SYSTEM System (* System Configuration *)
  (* Version 0.0, 7/6/2026, Schneider Electric *)
  APPLICATION Hidryco_Application
    (* CLP SUBSTACAO *)
    (* CLP NEREDA *)
    (* NEREDA REACTORS *)
    (* NEREDA PROCESS - HIDRYCO *)
    (* EMERGENCY RECIPIE *)
    (* NEREDA EQUIPMENT *)
    (* NEREDA AERATION *)
    (* INFLUENT FEED *)
    (* EFFLUENT *)
    (* SLUDGE BUFFER *)
    (* METAL SALT DOSING *)
    (* SLUDGE HOLDING TANK *)
    FBS
      A3_DI32K0 : IO_DI32(pin_46CCA44197086456 := '$${PATH}A3_DI32K_WORD0', pin_0CD1E891B208CBDA := '$${PATH}A3_DI32K_WORD1', pin_36419F0327C5E289 := 'RES0.InfluentFeed.Actuators.FeedReactorPump01.LocalPanel.SafetySwitchOff', pin_EB713021CCA66C0B := 'RES0.InfluentFeed.Actuators.FeedReactorPump02.LocalPanel.SafetySwitchOff', pin_2B28AC3EFC010509 := 'RES0.InfluentFeed.Actuators.FeedReactorPump03.LocalPanel.SafetySwitchOff', pin_ECB70C50847C6B8C := 'RES0.InfluentFeed.Actuators.FeedReactorPump01.LocalPanel.RemoteSelect', pin_07613AEA5B5EA3D4 := 'RES0.InfluentFeed.Actuators.FeedReactorPump01.fbFwd.DIn', pin_255156C9E2C187C7 := 'RES0.InfluentFeed.Actuators.FeedReactorPump01.LocalPanel.ElectricCircuitFail', pin_A4FEA1DCF2974931 := 'RES0.InfluentFeed.Actuators.FeedReactorPump01.LocalPanel.MoistureDetectionPumpMS', pin_330A6B5BAE9F40D2 := 'RES0.InfluentFeed.Actuators.FeedReactorPump02.LocalPanel.RemoteSelect', pin_15A3E3BB9AE8E740 := 'RES0.InfluentFeed.Actuators.FeedReactorPump02.fbFwd.DIn', pin_6F381A44E74CF961 := 'RES0.InfluentFeed.Actuators.FeedReactorPump02.LocalPanel.ElectricCircuitFail', pin_28174C1DE6948A82 := 'RES0.InfluentFeed.Actuators.FeedReactorPump02.LocalPanel.MoistureDetectionPumpMS', pin_1BA632E0922A0983 := 'RES0.InfluentFeed.Actuators.FeedReactorPump03.LocalPanel.RemoteSelect', pin_3F9A9A7D3F756840 := 'RES0.InfluentFeed.Actuators.FeedReactorPump03.fbFwd.DIn', pin_7C7DB6F90D480DE8 := 'RES0.InfluentFeed.Actuators.FeedReactorPump03.LocalPanel.ElectricCircuitFail', pin_E8D93A7BE9BA26AB := 'RES0.InfluentFeed.Actuators.FeedReactorPump03.LocalPanel.MoistureDetectionPumpMS', pin_2C3BA8CD03BB1AD1 := 'RES0.InfluentFeed.Actuators.Mixer01.LocalPanel.PowerFb', pin_BD4DD77DC1DECA3F := 'RES0.InfluentFeed.Actuators.Mixer02.LocalPanel.PowerFb', pin_BA2C5E15436FD50A := 'RES0.InfluentFeed.Actuators.Mixer01.LocalPanel.RemoteSelect', pin_58F1D1C70BD05BBB := 'RES0.InfluentFeed.Actuators.Mixer01.fbFwd.DIn', pin_202E08C1E95489B4 := 'RES0.InfluentFeed.Actuators.Mixer01.LocalPanel.ElectricCircuitFail', pin_4D7EBC78C81E0547 := 'RES0.InfluentFeed.Actuators.Mixer01.LocalPanel.MoistureDetectionPumpMS', pin_705DA0BDD5247341 := 'RES0.InfluentFeed.Actuators.Mixer02.LocalPanel.RemoteSelect', pin_C8A2275FCD06007F := 'RES0.InfluentFeed.Actuators.Mixer02.fbFwd.DIn', pin_029A065AE8EEF4A5 := '$${PATH}A3_DI32K0_CONN');
      A4_DI32K0 : IO_DI32(pin_46CCA44197086456 := '$${PATH}A4_DI32K_WORD0', pin_0CD1E891B208CBDA := '$${PATH}A4_DI32K_WORD1', pin_21F6274CBA1014D4 := 'RES0.InfluentFeed.Actuators.Mixer02.LocalPanel.ElectricCircuitFail', pin_828C0F18BDE4203E := 'RES0.InfluentFeed.Actuators.Mixer02.LocalPanel.MoistureDetectionPumpMS', pin_9E5CF06E07A0EB03 := 'RES0.SludgeBuffer.Actuators.Pump1.LocalPanel.PowerFb', pin_36419F0327C5E289 := 'RES0.SludgeBuffer.Actuators.Pump2.LocalPanel.PowerFb', pin_EB713021CCA66C0B := 'RES0.SludgeBuffer.Actuators.Pump3.LocalPanel.PowerFb', pin_2B28AC3EFC010509 := 'RES0.SludgeBuffer.Actuators.Pump1.LocalPanel.RemoteSelect', pin_ECB70C50847C6B8C := 'RES0.SludgeBuffer.Actuators.Pump1.fbFwd.DIn', pin_4067F611C03C22ED := 'RES0.SludgeBuffer.Actuators.Pump1.LocalPanel.ElectricCircuitFail', pin_07613AEA5B5EA3D4 := 'RES0.SludgeBuffer.Actuators.Pump2.LocalPanel.RemoteSelect', pin_A4FEA1DCF2974931 := 'RES0.SludgeBuffer.Actuators.Pump2.fbFwd.DIn', pin_330A6B5BAE9F40D2 := 'RES0.SludgeBuffer.Actuators.Pump2.LocalPanel.ElectricCircuitFail', pin_341ABC323332EA3F := 'RES0.SludgeBuffer.Actuators.Pump3.LocalPanel.RemoteSelect', pin_6F381A44E74CF961 := 'RES0.SludgeBuffer.Actuators.Pump3.fbFwd.DIn', pin_28174C1DE6948A82 := 'RES0.SludgeBuffer.Actuators.Pump3.LocalPanel.ElectricCircuitFail', pin_7C7DB6F90D480DE8 := 'RES0.Reactor1.Actuators.VentAerationGridValve_AV4x107.fbOpen.DIn', pin_E8D93A7BE9BA26AB := 'RES0.Reactor1.Actuators.VentAerationGridValve_AV4x107.fbClose.DIn', pin_2C3BA8CD03BB1AD1 := 'RES0.Reactor1.Actuators.AirFillValveSludgeDischarge_AV4x171.fbOpen.DIn', pin_BD4DD77DC1DECA3F := 'RES0.Reactor1.Actuators.AirFillValveSludgeDischarge_AV4x171.fbClose.DIn', pin_BA2C5E15436FD50A := 'RES0.Reactor1.Actuators.VentSludgeGridValve_AV4x172.fbOpen.DIn', pin_2DD13C1C321F4353 := 'RES0.Reactor1.Actuators.VentSludgeGridValve_AV4x172.fbClose.DIn', pin_58F1D1C70BD05BBB := 'RES0.Reactor1.Actuators.FeedValve_AV4x101.fbOpen.DIn', pin_202E08C1E95489B4 := 'RES0.Reactor1.Actuators.FeedValve_AV4x101.fbClose.DIn', pin_4D7EBC78C81E0547 := 'RES0.Reactor1.Actuators.LowerLevelValve_AV4x102.fbOpen.DIn', pin_705DA0BDD5247341 := 'RES0.Reactor1.Actuators.LowerLevelValve_AV4x102.fbClose.DIn', pin_3B4E2202D2B578AA := 'RES0.Reactor1.Actuators.DischargeValve_AV4x103.fbOpen.DIn', pin_C8A2275FCD06007F := 'RES0.Reactor1.Actuators.DischargeValve_AV4x103.fbClose.DIn', pin_029A065AE8EEF4A5 := 'RES0.A3_DI32K0.A3_DI32K0_CONN');
      A5_DI32K0 : IO_DI32(pin_46CCA44197086456 := '$${PATH}A5_DI32K_WORD0', pin_0CD1E891B208CBDA := '$${PATH}A5_DI32K_WORD1', pin_21F6274CBA1014D4 := 'RES0.Reactor2.Actuators.VentAerationGridValve_AV4x107.fbOpen.DIn', pin_828C0F18BDE4203E := 'RES0.Reactor2.Actuators.VentAerationGridValve_AV4x107.fbClose.DIn', pin_9E5CF06E07A0EB03 := 'RES0.Reactor2.Actuators.AirFillValveSludgeDischarge_AV4x171.fbOpen.DIn', pin_36419F0327C5E289 := 'RES0.Reactor2.Actuators.AirFillValveSludgeDischarge_AV4x171.fbClose.DIn', pin_EB713021CCA66C0B := 'RES0.Reactor2.Actuators.VentSludgeGridValve_AV4x172.fbOpen.DIn', pin_2B28AC3EFC010509 := 'RES0.Reactor2.Actuators.VentSludgeGridValve_AV4x172.fbClose.DIn', pin_772061FB1EC77CFC := 'RES0.Reactor2.Actuators.FeedValve_AV4x101.fbOpen.DIn', pin_ECB70C50847C6B8C := 'RES0.Reactor2.Actuators.FeedValve_AV4x101.fbClose.DIn', pin_4067F611C03C22ED := 'RES0.Reactor2.Actuators.LowerLevelValve_AV4x102.fbOpen.DIn', pin_07613AEA5B5EA3D4 := 'RES0.Reactor2.Actuators.LowerLevelValve_AV4x102.fbClose.DIn', pin_255156C9E2C187C7 := 'RES0.Reactor2.Actuators.DischargeValve_AV4x103.fbOpen.DIn', pin_A4FEA1DCF2974931 := 'RES0.Reactor2.Actuators.DischargeValve_AV4x103.fbClose.DIn', pin_15A3E3BB9AE8E740 := 'RES0.SludgeBuffer.Actuators.ValveBuffer.fbOpen.DIn', pin_6F381A44E74CF961 := 'RES0.SludgeBuffer.Actuators.ValveBuffer.fbClose.DIn', pin_28174C1DE6948A82 := 'RES0.SludgeBuffer.Actuators.ValveInfeed.fbOpen.DIn', pin_1BA632E0922A0983 := 'RES0.SludgeBuffer.Actuators.ValveInfeed.fbClose.DIn', pin_2C3BA8CD03BB1AD1 := 'RES0.InfluentFeed.Sensors.LevelSwitchInfluentBuffer.pv.DIn', pin_BD4DD77DC1DECA3F := 'RES0.Reactor1.Actuators.AerationBlockValve_AV4x170.fbOpen.DIn', pin_BA2C5E15436FD50A := 'RES0.Reactor1.Actuators.AerationBlockValve_AV4x170.fbClose.DIn', pin_2DD13C1C321F4353 := 'RES0.Reactor2.Actuators.AerationBlockValve_AV4x170.fbOpen.DIn', pin_58F1D1C70BD05BBB := 'RES0.Reactor2.Actuators.AerationBlockValve_AV4x170.fbClose.DIn', pin_029A065AE8EEF4A5 := 'RES0.A3_DI32K0.A3_DI32K0_CONN', pin_330A6B5BAE9F40D2 := 'RES0.SludgeBuffer.Actuators.ValveSupernatantReturn.fbOpen.DIn', pin_341ABC323332EA3F := 'RES0.SludgeBuffer.Actuators.ValveSupernatantReturn.fbClose.DIn', pin_23FCAB00EAAA7E55 := 'RES0.SludgeBuffer.Actuators.ValveTank2.fbOpen.DIn', pin_3F9A9A7D3F756840 := 'RES0.SludgeBuffer.Actuators.ValveTank2.fbClose.DIn', pin_7C7DB6F90D480DE8 := 'RES0.SludgeBuffer.Actuators.ValveTank1.fbOpen.DIn', pin_E8D93A7BE9BA26AB := 'RES0.SludgeBuffer.Actuators.ValveTank1.fbClose.DIn');
      A6_DI32K0 : IO_DI32(pin_46CCA44197086456 := '$${PATH}A6_DI32K_WORD0', pin_0CD1E891B208CBDA := '$${PATH}A6_DI32K_WORD1', pin_029A065AE8EEF4A5 := 'RES0.A3_DI32K0.A3_DI32K0_CONN');
      A7_DQ32TK0 : IO_DQ32(pin_302C3F69182ABC91 := '$${PATH}A7_DQ32TK_WORD0', pin_449EC30B868089F7 := '$${PATH}A7_DQ32TK_WORD1', pin_9A3A1A81B7B6D445 := 'RES0.InfluentFeed.Actuators.FeedReactorPump01.cmdFwd.DOut', pin_574F19B312039273 := 'RES0.InfluentFeed.Actuators.FeedReactorPump01.LocalPanel.ResetError_ATV', pin_289462D1695B79B9 := 'RES0.InfluentFeed.Actuators.FeedReactorPump02.cmdFwd.DOut', pin_312C400F6E937723 := 'RES0.InfluentFeed.Actuators.FeedReactorPump02.LocalPanel.ResetError_ATV', pin_3BE637AB2D7945FF := 'RES0.InfluentFeed.Actuators.FeedReactorPump03.cmdFwd.DOut', pin_22A55DF5D197312F := 'RES0.InfluentFeed.Actuators.FeedReactorPump03.LocalPanel.ResetError_ATV', pin_8561E9473423D106 := 'RES0.InfluentFeed.Actuators.Mixer01.cmdFwd.DOut', pin_22A9D026EB73BE1F := 'RES0.InfluentFeed.Actuators.Mixer01.LocalPanel.ResetError_ATV', pin_FA96DB2F4BA1237E := 'RES0.InfluentFeed.Actuators.Mixer02.cmdFwd.DOut', pin_29C78CF381382FF2 := 'RES0.InfluentFeed.Actuators.Mixer02.LocalPanel.ResetError_ATV', pin_29CEA3759F3752DE := 'RES0.SludgeBuffer.Actuators.Pump1.cmdFwd.DOut', pin_886E7CBF7859CEF7 := 'RES0.SludgeBuffer.Actuators.Pump1.LocalPanel.ResetError_ATV', pin_FD4664BC008BF5D6 := 'RES0.SludgeBuffer.Actuators.Pump2.cmdFwd.DOut', pin_33252EF2B10EEA13 := 'RES0.SludgeBuffer.Actuators.Pump2.LocalPanel.ResetError_ATV', pin_0AA04E78B7312E60 := 'RES0.SludgeBuffer.Actuators.Pump3.cmdFwd.DOut', pin_753BEBC4FB000D5B := 'RES0.SludgeBuffer.Actuators.Pump3.LocalPanel.ResetError_ATV', pin_9E16F3DA85027DF7 := 'RES0.Reactor1.Actuators.VentAerationGridValve_AV4x107.cmdOpen.DOut', pin_3452F813357567DB := 'RES0.Reactor1.Actuators.VentAerationGridValve_AV4x107.cmdClose.DOut', pin_19CF596687475EFF := 'RES0.Reactor1.Actuators.AirFillValveSludgeDischarge_AV4x171.cmdOpen.DOut', pin_894AD674E7043530 := 'RES0.Reactor1.Actuators.AirFillValveSludgeDischarge_AV4x171.cmdClose.DOut', pin_4C1794B9AC53DE50 := 'RES0.Reactor1.Actuators.VentSludgeGridValve_AV4x172.cmdOpen.DOut', pin_B27C16F31DA61BFA := 'RES0.Reactor1.Actuators.VentSludgeGridValve_AV4x172.cmdClose.DOut', pin_6AEF80E82895335D := 'RES0.Reactor1.Actuators.FeedValve_AV4x101.cmdOpen.DOut', pin_4CE944D399950301 := 'RES0.Reactor1.Actuators.FeedValve_AV4x101.cmdClose.DOut', pin_4A5E1556A870DE8E := 'RES0.Reactor1.Actuators.LowerLevelValve_AV4x102.cmdOpen.DOut', pin_BB019F781B1BA10A := 'RES0.Reactor1.Actuators.LowerLevelValve_AV4x102.cmdClose.DOut', pin_86F66632C3A9C16C := 'RES0.Reactor1.Actuators.DischargeValve_AV4x103.cmdOpen.DOut', pin_B6D2486BB09D13CD := 'RES0.Reactor1.Actuators.DischargeValve_AV4x103.cmdClose.DOut', pin_51993B782C6727EF := 'RES0.Reactor2.Actuators.VentAerationGridValve_AV4x107.cmdOpen.DOut', pin_C59E5F7297A9D375 := 'RES0.Reactor2.Actuators.VentAerationGridValve_AV4x107.cmdClose.DOut', pin_713D841585687888 := 'RES0.Reactor2.Actuators.AirFillValveSludgeDischarge_AV4x171.cmdOpen.DOut', pin_F178B2FCFCB541E9 := 'RES0.Reactor2.Actuators.AirFillValveSludgeDischarge_AV4x171.cmdClose.DOut', pin_4CB528AC475AE599 := 'RES0.A3_DI32K0.A3_DI32K0_CONN');
      A8_DQ32TK0 : IO_DQ32(pin_302C3F69182ABC91 := '$${PATH}A8_DQ32TK_WORD0', pin_449EC30B868089F7 := '$${PATH}A8_DQ32TK_WORD1', pin_9A3A1A81B7B6D445 := 'RES0.Reactor2.Actuators.VentSludgeGridValve_AV4x172.cmdOpen.DOut', pin_574F19B312039273 := 'RES0.Reactor2.Actuators.VentSludgeGridValve_AV4x172.cmdClose.DOut', pin_289462D1695B79B9 := 'RES0.Reactor2.Actuators.FeedValve_AV4x101.cmdOpen.DOut', pin_312C400F6E937723 := 'RES0.Reactor2.Actuators.FeedValve_AV4x101.cmdClose.DOut', pin_3BE637AB2D7945FF := 'RES0.Reactor2.Actuators.LowerLevelValve_AV4x102.cmdOpen.DOut', pin_22A55DF5D197312F := 'RES0.Reactor2.Actuators.LowerLevelValve_AV4x102.cmdClose.DOut', pin_8561E9473423D106 := 'RES0.Reactor2.Actuators.DischargeValve_AV4x103.cmdOpen.DOut', pin_22A9D026EB73BE1F := 'RES0.Reactor2.Actuators.DischargeValve_AV4x103.cmdClose.DOut', pin_29CEA3759F3752DE := 'RES0.SludgeBuffer.Actuators.ValveBuffer.cmdOpen.DOut', pin_886E7CBF7859CEF7 := 'RES0.SludgeBuffer.Actuators.ValveBuffer.cmdClose.DOut', pin_FD4664BC008BF5D6 := 'RES0.SludgeBuffer.Actuators.ValveInfeed.cmdOpen.DOut', pin_33252EF2B10EEA13 := 'RES0.SludgeBuffer.Actuators.ValveInfeed.cmdClose.DOut', pin_19CF596687475EFF := 'RES0.Reactor1.Actuators.AerationBlockValve_AV4x170.cmdOpen.DOut', pin_894AD674E7043530 := 'RES0.Reactor1.Actuators.AerationBlockValve_AV4x170.cmdClose.DOut', pin_4C1794B9AC53DE50 := 'RES0.Reactor2.Actuators.AerationBlockValve_AV4x170.cmdOpen.DOut', pin_B27C16F31DA61BFA := 'RES0.Reactor2.Actuators.AerationBlockValve_AV4x170.cmdClose.DOut', pin_4CB528AC475AE599 := 'RES0.A3_DI32K0.A3_DI32K0_CONN', pin_FA96DB2F4BA1237E := 'RES0.SludgeBuffer.Actuators.ValveSupernatantReturn.cmdOpen.DOut', pin_29C78CF381382FF2 := 'RES0.SludgeBuffer.Actuators.ValveSupernatantReturn.cmdClose.DOut', pin_3452F813357567DB := 'RES0.SludgeBuffer.Actuators.ValveTank1.cmdClose.DOut', pin_9E16F3DA85027DF7 := 'RES0.SludgeBuffer.Actuators.ValveTank1.cmdOpen.DOut', pin_0AA04E78B7312E60 := 'RES0.SludgeBuffer.Actuators.ValveTank2.cmdOpen.DOut', pin_753BEBC4FB000D5B := 'RES0.SludgeBuffer.Actuators.ValveTank2.cmdClose.DOut');
      SUB_A3_DI32K0 : IO_DI32(pin_46CCA44197086456 := '$${PATH}SUB_A3_DI32K_WORD0', pin_0CD1E891B208CBDA := '$${PATH}SUB_A3_DI32K_WORD1', pin_23FCAB00EAAA7E55 := 'RES0.Aerator.Actuators.V4603.LocalPanel.PowerFb', pin_3F9A9A7D3F756840 := 'RES0.Aerator.Actuators.V4604.LocalPanel.PowerFb', pin_029A065AE8EEF4A5 := '$${PATH}SUB_A3_DI32K0_CONN');
      SUB_A4_DI32K0 : IO_DI32(pin_46CCA44197086456 := '$${PATH}SUB_A4_DI32K_WORD0', pin_0CD1E891B208CBDA := '$${PATH}SUB_A4_DI32K_WORD1', pin_3B4E2202D2B578AA := 'RES0.Aerator.Actuators.V4601.LocalPanel.PowerFb', pin_C8A2275FCD06007F := 'RES0.Aerator.Actuators.V4602.LocalPanel.PowerFb', pin_029A065AE8EEF4A5 := 'RES0.SUB_A3_DI32K0.SUB_A3_DI32K0_CONN');
      SUB_A6_DI32K0 : IO_DI32(pin_46CCA44197086456 := '$${PATH}SUB_A6_DI32K_WORD0', pin_0CD1E891B208CBDA := '$${PATH}SUB_A6_DI32K_WORD1', pin_255156C9E2C187C7 := 'RES0.Aerator.Actuators.AV46_001.fbOpen.DIn', pin_A4FEA1DCF2974931 := 'RES0.Aerator.Actuators.AV46_001.fbClose.DIn', pin_330A6B5BAE9F40D2 := 'RES0.Aerator.Actuators.AV46_002.fbOpen.DIn', pin_341ABC323332EA3F := 'RES0.Aerator.Actuators.AV46_002.fbClose.DIn', pin_15A3E3BB9AE8E740 := 'RES0.Aerator.Actuators.AV46_003.fbOpen.DIn', pin_6F381A44E74CF961 := 'RES0.Aerator.Actuators.AV46_003.fbClose.DIn', pin_28174C1DE6948A82 := 'RES0.Aerator.Actuators.AV46_012.fbOpen.DIn', pin_1BA632E0922A0983 := 'RES0.Aerator.Actuators.AV46_012.fbClose.DIn', pin_23FCAB00EAAA7E55 := 'RES0.Aerator.Actuators.AV46_022.fbOpen.DIn', pin_3F9A9A7D3F756840 := 'RES0.Aerator.Actuators.AV46_022.fbClose.DIn', pin_7C7DB6F90D480DE8 := 'RES0.Aerator.Actuators.AV46_032.fbOpen.DIn', pin_E8D93A7BE9BA26AB := 'RES0.Aerator.Actuators.AV46_032.fbClose.DIn', pin_2C3BA8CD03BB1AD1 := 'RES0.Aerator.Actuators.AV46_042.fbOpen.DIn', pin_BD4DD77DC1DECA3F := 'RES0.Aerator.Actuators.AV46_042.fbClose.DIn', pin_029A065AE8EEF4A5 := 'RES0.SUB_A3_DI32K0.SUB_A3_DI32K0_CONN');
      SUB_A8_DQ32TK0 : IO_DQ32(pin_302C3F69182ABC91 := '$${PATH}SUB_A8_DQ32TK_WORD0', pin_449EC30B868089F7 := '$${PATH}SUB_A8_DQ32TK_WORD1', pin_19CF596687475EFF := 'RES0.Aerator.Actuators.AV46_001.cmdOpen.DOut', pin_894AD674E7043530 := 'RES0.Aerator.Actuators.AV46_001.cmdClose.DOut', pin_4C1794B9AC53DE50 := 'RES0.Aerator.Actuators.AV46_002.cmdOpen.DOut', pin_B27C16F31DA61BFA := 'RES0.Aerator.Actuators.AV46_002.cmdClose.DOut', pin_6AEF80E82895335D := 'RES0.Aerator.Actuators.AV46_003.cmdOpen.DOut', pin_4CE944D399950301 := 'RES0.Aerator.Actuators.AV46_003.cmdClose.DOut', pin_4A5E1556A870DE8E := 'RES0.Aerator.Actuators.AV46_012.cmdOpen.DOut', pin_BB019F781B1BA10A := 'RES0.Aerator.Actuators.AV46_012.cmdClose.DOut', pin_86F66632C3A9C16C := 'RES0.Aerator.Actuators.AV46_022.cmdOpen.DOut', pin_B6D2486BB09D13CD := 'RES0.Aerator.Actuators.AV46_022.cmdClose.DOut', pin_51993B782C6727EF := 'RES0.Aerator.Actuators.AV46_032.cmdOpen.DOut', pin_C59E5F7297A9D375 := 'RES0.Aerator.Actuators.AV46_032.cmdClose.DOut', pin_713D841585687888 := 'RES0.Aerator.Actuators.AV46_042.cmdOpen.DOut', pin_F178B2FCFCB541E9 := 'RES0.Aerator.Actuators.AV46_042.cmdClose.DOut', pin_4CB528AC475AE599 := 'RES0.SUB_A3_DI32K0.SUB_A3_DI32K0_CONN');
      V4601_STS0 : IO_DI32(pin_46CCA44197086456 := '$${PATH}V4601_STATUS', pin_0CD1E891B208CBDA := '$${PATH}V4601_FAULT', pin_029A065AE8EEF4A5 := '$${PATH}V4601_CONN', pin_21F6274CBA1014D4 := 'RES0.Aerator.Actuators.V4601.LocalPanel.RemoteSelect', pin_828C0F18BDE4203E := 'RES0.Aerator.Actuators.V4601.fbFwd.DIn', pin_36419F0327C5E289 := 'RES0.Aerator.Actuators.V4601.LocalPanel.FrequencyInverterFail', pin_4067F611C03C22ED := 'RES0.Aerator.Actuators.V4601.LocalPanel.AtvReady');
      V4601_CMD0 : IO_DQ32(pin_302C3F69182ABC91 := '$${PATH}V4601_CMD_WORD', pin_449EC30B868089F7 := '$${PATH}V4601_WORD1_NAO_USADA', pin_9A3A1A81B7B6D445 := 'RES0.Aerator.Actuators.V4601.cmdFwd.DOut', pin_289462D1695B79B9 := 'RES0.Aerator.Actuators.V4601.LocalPanel.ResetError_ATV');
      V4602_STS0 : IO_DI32(pin_46CCA44197086456 := '$${PATH}V4602_STATUS', pin_0CD1E891B208CBDA := '$${PATH}V4602_FAULT', pin_029A065AE8EEF4A5 := '$${PATH}V4602_CONN', pin_21F6274CBA1014D4 := 'RES0.Aerator.Actuators.V4602.LocalPanel.RemoteSelect', pin_828C0F18BDE4203E := 'RES0.Aerator.Actuators.V4602.fbFwd.DIn', pin_36419F0327C5E289 := 'RES0.Aerator.Actuators.V4602.LocalPanel.FrequencyInverterFail', pin_4067F611C03C22ED := 'RES0.Aerator.Actuators.V4602.LocalPanel.AtvReady');
      V4602_CMD0 : IO_DQ32(pin_302C3F69182ABC91 := '$${PATH}V4602_CMD_WORD', pin_449EC30B868089F7 := '$${PATH}V4602_WORD1_NAO_USADA', pin_9A3A1A81B7B6D445 := 'RES0.Aerator.Actuators.V4602.cmdFwd.DOut', pin_289462D1695B79B9 := 'RES0.Aerator.Actuators.V4602.LocalPanel.ResetError_ATV');
      V4603_STS0 : IO_DI32(pin_46CCA44197086456 := '$${PATH}V4603_STATUS', pin_0CD1E891B208CBDA := '$${PATH}V4603_FAULT', pin_029A065AE8EEF4A5 := '$${PATH}V4603_CONN', pin_21F6274CBA1014D4 := 'RES0.Aerator.Actuators.V4603.LocalPanel.RemoteSelect', pin_828C0F18BDE4203E := 'RES0.Aerator.Actuators.V4603.fbFwd.DIn', pin_36419F0327C5E289 := 'RES0.Aerator.Actuators.V4603.LocalPanel.FrequencyInverterFail', pin_4067F611C03C22ED := 'RES0.Aerator.Actuators.V4603.LocalPanel.AtvReady');
      V4603_CMD0 : IO_DQ32(pin_302C3F69182ABC91 := '$${PATH}V4603_CMD_WORD', pin_449EC30B868089F7 := '$${PATH}V4603_WORD1_NAO_USADA', pin_9A3A1A81B7B6D445 := 'RES0.Aerator.Actuators.V4603.cmdFwd.DOut', pin_289462D1695B79B9 := 'RES0.Aerator.Actuators.V4603.LocalPanel.ResetError_ATV');
      V4604_STS0 : IO_DI32(pin_46CCA44197086456 := '$${PATH}V4604_STATUS', pin_0CD1E891B208CBDA := '$${PATH}V4604_FAULT', pin_029A065AE8EEF4A5 := '$${PATH}V4604_CONN', pin_21F6274CBA1014D4 := 'RES0.Aerator.Actuators.V4604.LocalPanel.RemoteSelect', pin_828C0F18BDE4203E := 'RES0.Aerator.Actuators.V4604.fbFwd.DIn', pin_36419F0327C5E289 := 'RES0.Aerator.Actuators.V4604.LocalPanel.FrequencyInverterFail', pin_4067F611C03C22ED := 'RES0.Aerator.Actuators.V4604.LocalPanel.AtvReady');
      V4604_CMD0 : IO_DQ32(pin_302C3F69182ABC91 := '$${PATH}V4604_CMD_WORD', pin_449EC30B868089F7 := '$${PATH}V4604_WORD1_NAO_USADA', pin_9A3A1A81B7B6D445 := 'RES0.Aerator.Actuators.V4604.cmdFwd.DOut', pin_289462D1695B79B9 := 'RES0.Aerator.Actuators.V4604.LocalPanel.ResetError_ATV');
      Mode : Mode; {SET_ATTRIBUTE(CompilerOptions, CheckConnectionsStrictly=False)}
      OpenWebPage : OpenWebPage(URL := 'http://192.168.1.10');
      OTHERS_DISCHARGE_VALVES_FB : OthersDischargeValves;
      EmergencyManagement : EmergencyManagement;
      Utilities : Utilities;
      EnergySignal : Frequency_Power;
      HeartBeat1 : HeartBeat;
      Aerator : NeredaCAeration;
      SludgeBuffer : NeredaSludgeBuffer_2;
      SludgeHoldingTank1 : SludgeHoldingTank;
      SludgeHoldingTank2 : SludgeHoldingTank;
      Reactor1 : NeredaReactor;
      Reactor2 : NeredaReactor;
      EmergencySB : EmergencySludgeBuffer;
      EmergencyReactor1 : EmergencyReactor_2;
      EmergencyReactor2 : EmergencyReactor_2;
      InfluentFeed : InfluentFeed;
    END_FBS
    ADAPTER_CONNECTIONS
      HeartBeat1.40 TO Mode.6E012D59F948069E;
      Mode.50 TO SludgeBuffer.6D7943A09F73313C;
      InfluentFeed.06B5BF90025137D8 TO SludgeBuffer.04BD059D1BCDA8FF;
      InfluentFeed.08DA021DBE2FF670 TO SludgeBuffer.34E82C716D68805B;
      SludgeHoldingTank1.745E7C7F86CD93D6 TO SludgeBuffer.1369AAF8C65D025F;
      SludgeHoldingTank2.745E7C7F86CD93D6 TO SludgeBuffer.103390B72A3B733A;
      OTHERS_DISCHARGE_VALVES_FB.82A979F8A1C1CE4A TO Reactor1.AE9DB11716461BE5;
      OTHERS_DISCHARGE_VALVES_FB.00DDB30B96836B1C TO Reactor2.AE9DB11716461BE5;
      Mode.39 TO Reactor1.8E8BC8CAE0ABBEF0;
      Mode.40 TO Reactor2.8E8BC8CAE0ABBEF0;
      Mode.55 TO EmergencyManagement.FA37C5C7FF880AB4;
      Reactor1.53509993DCC2E69E TO EmergencyManagement.03E1DF24854B5087;
      Reactor2.53509993DCC2E69E TO EmergencyManagement.8D40980BCD10D06B;
      EmergencyManagement.5C1263F1F6F0F578 TO EmergencyReactor1.73503C83163B2D86;
      EmergencyManagement.6B6FC4EBFE551754 TO EmergencyReactor2.73503C83163B2D86;
      Reactor1.E962C7AC1C669349 TO Aerator.IBlowerReactor;
      Reactor2.E962C7AC1C669349 TO Aerator.036B0699AE92B07E;
      Reactor1.EF12C2F0857E0401 TO InfluentFeed.458126F8619187E9;
      Reactor2.EF12C2F0857E0401 TO InfluentFeed.13A00CB3B1B3C5BD;
      EmergencyReactor1.ADE9AC252194767E TO Reactor1.4FE3E9A63522A043;
      EmergencyReactor2.ADE9AC252194767E TO Reactor2.4FE3E9A63522A043;
      SludgeBuffer.5220CD4AB4D5EF57 TO Reactor1.64A5E847CFF537B2;
      SludgeBuffer.F8A56E33E99EA0E4 TO Reactor2.64A5E847CFF537B2;
      SludgeBuffer.2EF6B69B645AE6E1 TO InfluentFeed.9135BA3E72B25810;
      EmergencyManagement.10001B393681040B TO OTHERS_DISCHARGE_VALVES_FB.0FC638121CDA6752;
      SludgeBuffer.8B97DDD2DF3E853F TO EmergencyManagement.92B17EFA7CB0DA14;
      EmergencyReactor2.D6CF55AACA664FB9 TO EmergencySB.A9597B321AC24B8F;
      EmergencyReactor1.D6CF55AACA664FB9 TO EmergencySB.E201588BE0264C59;
      InfluentFeed.072EC58E32F5B902 TO Reactor1.9D6CC0A1E886795A;
      InfluentFeed.57887779F0B6E332 TO Reactor2.9D6CC0A1E886795A;
      SludgeBuffer.0CE6DD66A1C58D5B TO Reactor1.6D054A47338EC161;
      SludgeBuffer.DE069E6752438E1A TO Reactor2.6D054A47338EC161;
      EmergencySB.CC52284A3E90E837 TO SludgeBuffer.8642DEF89CD05FB2;
    END_CONNECTIONS
  END_APPLICATION
  DEVICE M262_Lodo : M262_dPAC
    RESOURCE RES0 : EMB_RES_ECO
    END_RESOURCE
  END_DEVICE
  DEVICE HMI2 : HMI_NET
  END_DEVICE
  DEVICE M262_Substacao : M262_dPAC
    RESOURCE RES0 : EMB_RES_ECO
    END_RESOURCE
  END_DEVICE
  DEVICE M262_Nereda : M262_dPAC
    RESOURCE RES0 : EMB_RES_ECO
      FBS
        DPAC_FULLINIT1 : DPAC_FULLINIT;
        OpenWebPage : OpenWebPage(URL := 'http://192.168.1.10');
        OTHERS_DISCHARGE_VALVES_FB : OthersDischargeValves;
        EmergencyManagement : EmergencyManagement;
        Utilities : Utilities;
        EnergySignal : Frequency_Power;
        HeartBeat1 : HeartBeat;
        Aerator : NeredaCAeration;
        SludgeBuffer : NeredaSludgeBuffer_2;
        EmergencyReactor1 : EmergencyReactor_2;
        EmergencyReactor2 : EmergencyReactor_2;
        Reactor2 : NeredaReactor;
        EmergencySB : EmergencySludgeBuffer;
        Reactor1 : NeredaReactor;
        Mode : Mode; {SET_ATTRIBUTE(CompilerOptions, CheckConnectionsStrictly=False)}
        InfluentFeed : InfluentFeed;
        A3_DI32K0 : IO_DI32(pin_46CCA44197086456 := '$${PATH}A3_DI32K_WORD0', pin_0CD1E891B208CBDA := '$${PATH}A3_DI32K_WORD1', pin_029A065AE8EEF4A5 := '$${PATH}A3_DI32K0_CONN', pin_36419F0327C5E289 := 'RES0.InfluentFeed.Actuators.FeedReactorPump01.LocalPanel.SafetySwitchOff', pin_EB713021CCA66C0B := 'RES0.InfluentFeed.Actuators.FeedReactorPump02.LocalPanel.SafetySwitchOff', pin_2B28AC3EFC010509 := 'RES0.InfluentFeed.Actuators.FeedReactorPump03.LocalPanel.SafetySwitchOff', pin_ECB70C50847C6B8C := 'RES0.InfluentFeed.Actuators.FeedReactorPump01.LocalPanel.RemoteSelect', pin_07613AEA5B5EA3D4 := 'RES0.InfluentFeed.Actuators.FeedReactorPump01.fbFwd.DIn', pin_255156C9E2C187C7 := 'RES0.InfluentFeed.Actuators.FeedReactorPump01.LocalPanel.ElectricCircuitFail', pin_A4FEA1DCF2974931 := 'RES0.InfluentFeed.Actuators.FeedReactorPump01.LocalPanel.MoistureDetectionPumpMS', pin_330A6B5BAE9F40D2 := 'RES0.InfluentFeed.Actuators.FeedReactorPump02.LocalPanel.RemoteSelect', pin_15A3E3BB9AE8E740 := 'RES0.InfluentFeed.Actuators.FeedReactorPump02.fbFwd.DIn', pin_6F381A44E74CF961 := 'RES0.InfluentFeed.Actuators.FeedReactorPump02.LocalPanel.ElectricCircuitFail', pin_28174C1DE6948A82 := 'RES0.InfluentFeed.Actuators.FeedReactorPump02.LocalPanel.MoistureDetectionPumpMS', pin_1BA632E0922A0983 := 'RES0.InfluentFeed.Actuators.FeedReactorPump03.LocalPanel.RemoteSelect', pin_3F9A9A7D3F756840 := 'RES0.InfluentFeed.Actuators.FeedReactorPump03.fbFwd.DIn', pin_7C7DB6F90D480DE8 := 'RES0.InfluentFeed.Actuators.FeedReactorPump03.LocalPanel.ElectricCircuitFail', pin_E8D93A7BE9BA26AB := 'RES0.InfluentFeed.Actuators.FeedReactorPump03.LocalPanel.MoistureDetectionPumpMS', pin_2C3BA8CD03BB1AD1 := 'RES0.InfluentFeed.Actuators.Mixer01.LocalPanel.PowerFb', pin_BD4DD77DC1DECA3F := 'RES0.InfluentFeed.Actuators.Mixer02.LocalPanel.PowerFb', pin_BA2C5E15436FD50A := 'RES0.InfluentFeed.Actuators.Mixer01.LocalPanel.RemoteSelect', pin_58F1D1C70BD05BBB := 'RES0.InfluentFeed.Actuators.Mixer01.fbFwd.DIn', pin_202E08C1E95489B4 := 'RES0.InfluentFeed.Actuators.Mixer01.LocalPanel.ElectricCircuitFail', pin_4D7EBC78C81E0547 := 'RES0.InfluentFeed.Actuators.Mixer01.LocalPanel.MoistureDetectionPumpMS', pin_705DA0BDD5247341 := 'RES0.InfluentFeed.Actuators.Mixer02.LocalPanel.RemoteSelect', pin_C8A2275FCD06007F := 'RES0.InfluentFeed.Actuators.Mixer02.fbFwd.DIn');
        A4_DI32K0 : IO_DI32(pin_46CCA44197086456 := '$${PATH}A4_DI32K_WORD0', pin_0CD1E891B208CBDA := '$${PATH}A4_DI32K_WORD1', pin_029A065AE8EEF4A5 := 'RES0.A3_DI32K0.A3_DI32K0_CONN', pin_21F6274CBA1014D4 := 'RES0.InfluentFeed.Actuators.Mixer02.LocalPanel.ElectricCircuitFail', pin_828C0F18BDE4203E := 'RES0.InfluentFeed.Actuators.Mixer02.LocalPanel.MoistureDetectionPumpMS', pin_9E5CF06E07A0EB03 := 'RES0.SludgeBuffer.Actuators.Pump1.LocalPanel.PowerFb', pin_36419F0327C5E289 := 'RES0.SludgeBuffer.Actuators.Pump2.LocalPanel.PowerFb', pin_EB713021CCA66C0B := 'RES0.SludgeBuffer.Actuators.Pump3.LocalPanel.PowerFb', pin_2B28AC3EFC010509 := 'RES0.SludgeBuffer.Actuators.Pump1.LocalPanel.RemoteSelect', pin_ECB70C50847C6B8C := 'RES0.SludgeBuffer.Actuators.Pump1.fbFwd.DIn', pin_4067F611C03C22ED := 'RES0.SludgeBuffer.Actuators.Pump1.LocalPanel.ElectricCircuitFail', pin_07613AEA5B5EA3D4 := 'RES0.SludgeBuffer.Actuators.Pump2.LocalPanel.RemoteSelect', pin_A4FEA1DCF2974931 := 'RES0.SludgeBuffer.Actuators.Pump2.fbFwd.DIn', pin_330A6B5BAE9F40D2 := 'RES0.SludgeBuffer.Actuators.Pump2.LocalPanel.ElectricCircuitFail', pin_341ABC323332EA3F := 'RES0.SludgeBuffer.Actuators.Pump3.LocalPanel.RemoteSelect', pin_6F381A44E74CF961 := 'RES0.SludgeBuffer.Actuators.Pump3.fbFwd.DIn', pin_28174C1DE6948A82 := 'RES0.SludgeBuffer.Actuators.Pump3.LocalPanel.ElectricCircuitFail', pin_7C7DB6F90D480DE8 := 'RES0.Reactor1.Actuators.VentAerationGridValve_AV4x107.fbOpen.DIn', pin_E8D93A7BE9BA26AB := 'RES0.Reactor1.Actuators.VentAerationGridValve_AV4x107.fbClose.DIn', pin_2C3BA8CD03BB1AD1 := 'RES0.Reactor1.Actuators.AirFillValveSludgeDischarge_AV4x171.fbOpen.DIn', pin_BD4DD77DC1DECA3F := 'RES0.Reactor1.Actuators.AirFillValveSludgeDischarge_AV4x171.fbClose.DIn', pin_BA2C5E15436FD50A := 'RES0.Reactor1.Actuators.VentSludgeGridValve_AV4x172.fbOpen.DIn', pin_2DD13C1C321F4353 := 'RES0.Reactor1.Actuators.VentSludgeGridValve_AV4x172.fbClose.DIn', pin_58F1D1C70BD05BBB := 'RES0.Reactor1.Actuators.FeedValve_AV4x101.fbOpen.DIn', pin_202E08C1E95489B4 := 'RES0.Reactor1.Actuators.FeedValve_AV4x101.fbClose.DIn', pin_4D7EBC78C81E0547 := 'RES0.Reactor1.Actuators.LowerLevelValve_AV4x102.fbOpen.DIn', pin_705DA0BDD5247341 := 'RES0.Reactor1.Actuators.LowerLevelValve_AV4x102.fbClose.DIn', pin_3B4E2202D2B578AA := 'RES0.Reactor1.Actuators.DischargeValve_AV4x103.fbOpen.DIn', pin_C8A2275FCD06007F := 'RES0.Reactor1.Actuators.DischargeValve_AV4x103.fbClose.DIn');
        A5_DI32K0 : IO_DI32(pin_46CCA44197086456 := '$${PATH}A5_DI32K_WORD0', pin_0CD1E891B208CBDA := '$${PATH}A5_DI32K_WORD1', pin_029A065AE8EEF4A5 := 'RES0.A3_DI32K0.A3_DI32K0_CONN', pin_21F6274CBA1014D4 := 'RES0.Reactor2.Actuators.VentAerationGridValve_AV4x107.fbOpen.DIn', pin_828C0F18BDE4203E := 'RES0.Reactor2.Actuators.VentAerationGridValve_AV4x107.fbClose.DIn', pin_9E5CF06E07A0EB03 := 'RES0.Reactor2.Actuators.AirFillValveSludgeDischarge_AV4x171.fbOpen.DIn', pin_36419F0327C5E289 := 'RES0.Reactor2.Actuators.AirFillValveSludgeDischarge_AV4x171.fbClose.DIn', pin_EB713021CCA66C0B := 'RES0.Reactor2.Actuators.VentSludgeGridValve_AV4x172.fbOpen.DIn', pin_2B28AC3EFC010509 := 'RES0.Reactor2.Actuators.VentSludgeGridValve_AV4x172.fbClose.DIn', pin_772061FB1EC77CFC := 'RES0.Reactor2.Actuators.FeedValve_AV4x101.fbOpen.DIn', pin_ECB70C50847C6B8C := 'RES0.Reactor2.Actuators.FeedValve_AV4x101.fbClose.DIn', pin_4067F611C03C22ED := 'RES0.Reactor2.Actuators.LowerLevelValve_AV4x102.fbOpen.DIn', pin_07613AEA5B5EA3D4 := 'RES0.Reactor2.Actuators.LowerLevelValve_AV4x102.fbClose.DIn', pin_255156C9E2C187C7 := 'RES0.Reactor2.Actuators.DischargeValve_AV4x103.fbOpen.DIn', pin_A4FEA1DCF2974931 := 'RES0.Reactor2.Actuators.DischargeValve_AV4x103.fbClose.DIn', pin_330A6B5BAE9F40D2 := 'RES0.SludgeBuffer.Actuators.ValveSupernatantReturn.fbOpen.DIn', pin_341ABC323332EA3F := 'RES0.SludgeBuffer.Actuators.ValveSupernatantReturn.fbClose.DIn', pin_15A3E3BB9AE8E740 := 'RES0.SludgeBuffer.Actuators.ValveBuffer.fbOpen.DIn', pin_6F381A44E74CF961 := 'RES0.SludgeBuffer.Actuators.ValveBuffer.fbClose.DIn', pin_28174C1DE6948A82 := 'RES0.SludgeBuffer.Actuators.ValveInfeed.fbOpen.DIn', pin_1BA632E0922A0983 := 'RES0.SludgeBuffer.Actuators.ValveInfeed.fbClose.DIn', pin_2C3BA8CD03BB1AD1 := 'RES0.InfluentFeed.Sensors.LevelSwitchInfluentBuffer.pv.DIn', pin_BD4DD77DC1DECA3F := 'RES0.Reactor1.Actuators.AerationBlockValve_AV4x170.fbOpen.DIn', pin_BA2C5E15436FD50A := 'RES0.Reactor1.Actuators.AerationBlockValve_AV4x170.fbClose.DIn', pin_2DD13C1C321F4353 := 'RES0.Reactor2.Actuators.AerationBlockValve_AV4x170.fbOpen.DIn', pin_58F1D1C70BD05BBB := 'RES0.Reactor2.Actuators.AerationBlockValve_AV4x170.fbClose.DIn', pin_23FCAB00EAAA7E55 := 'RES0.SludgeBuffer.Actuators.ValveTank2.fbOpen.DIn', pin_3F9A9A7D3F756840 := 'RES0.SludgeBuffer.Actuators.ValveTank2.fbClose.DIn', pin_7C7DB6F90D480DE8 := 'RES0.SludgeBuffer.Actuators.ValveTank1.fbOpen.DIn', pin_E8D93A7BE9BA26AB := 'RES0.SludgeBuffer.Actuators.ValveTank1.fbClose.DIn');
        A6_DI32K0 : IO_DI32(pin_46CCA44197086456 := '$${PATH}A6_DI32K_WORD0', pin_0CD1E891B208CBDA := '$${PATH}A6_DI32K_WORD1', pin_029A065AE8EEF4A5 := 'RES0.A3_DI32K0.A3_DI32K0_CONN');
        A7_DQ32TK0 : IO_DQ32(pin_302C3F69182ABC91 := '$${PATH}A7_DQ32TK_WORD0', pin_449EC30B868089F7 := '$${PATH}A7_DQ32TK_WORD1', pin_4CB528AC475AE599 := 'RES0.A3_DI32K0.A3_DI32K0_CONN', pin_9A3A1A81B7B6D445 := 'RES0.InfluentFeed.Actuators.FeedReactorPump01.cmdFwd.DOut', pin_574F19B312039273 := 'RES0.InfluentFeed.Actuators.FeedReactorPump01.LocalPanel.ResetError_ATV', pin_289462D1695B79B9 := 'RES0.InfluentFeed.Actuators.FeedReactorPump02.cmdFwd.DOut', pin_312C400F6E937723 := 'RES0.InfluentFeed.Actuators.FeedReactorPump02.LocalPanel.ResetError_ATV', pin_3BE637AB2D7945FF := 'RES0.InfluentFeed.Actuators.FeedReactorPump03.cmdFwd.DOut', pin_22A55DF5D197312F := 'RES0.InfluentFeed.Actuators.FeedReactorPump03.LocalPanel.ResetError_ATV', pin_8561E9473423D106 := 'RES0.InfluentFeed.Actuators.Mixer01.cmdFwd.DOut', pin_22A9D026EB73BE1F := 'RES0.InfluentFeed.Actuators.Mixer01.LocalPanel.ResetError_ATV', pin_FA96DB2F4BA1237E := 'RES0.InfluentFeed.Actuators.Mixer02.cmdFwd.DOut', pin_29C78CF381382FF2 := 'RES0.InfluentFeed.Actuators.Mixer02.LocalPanel.ResetError_ATV', pin_29CEA3759F3752DE := 'RES0.SludgeBuffer.Actuators.Pump1.cmdFwd.DOut', pin_886E7CBF7859CEF7 := 'RES0.SludgeBuffer.Actuators.Pump1.LocalPanel.ResetError_ATV', pin_FD4664BC008BF5D6 := 'RES0.SludgeBuffer.Actuators.Pump2.cmdFwd.DOut', pin_33252EF2B10EEA13 := 'RES0.SludgeBuffer.Actuators.Pump2.LocalPanel.ResetError_ATV', pin_0AA04E78B7312E60 := 'RES0.SludgeBuffer.Actuators.Pump3.cmdFwd.DOut', pin_753BEBC4FB000D5B := 'RES0.SludgeBuffer.Actuators.Pump3.LocalPanel.ResetError_ATV', pin_9E16F3DA85027DF7 := 'RES0.Reactor1.Actuators.VentAerationGridValve_AV4x107.cmdOpen.DOut', pin_3452F813357567DB := 'RES0.Reactor1.Actuators.VentAerationGridValve_AV4x107.cmdClose.DOut', pin_19CF596687475EFF := 'RES0.Reactor1.Actuators.AirFillValveSludgeDischarge_AV4x171.cmdOpen.DOut', pin_894AD674E7043530 := 'RES0.Reactor1.Actuators.AirFillValveSludgeDischarge_AV4x171.cmdClose.DOut', pin_4C1794B9AC53DE50 := 'RES0.Reactor1.Actuators.VentSludgeGridValve_AV4x172.cmdOpen.DOut', pin_B27C16F31DA61BFA := 'RES0.Reactor1.Actuators.VentSludgeGridValve_AV4x172.cmdClose.DOut', pin_6AEF80E82895335D := 'RES0.Reactor1.Actuators.FeedValve_AV4x101.cmdOpen.DOut', pin_4CE944D399950301 := 'RES0.Reactor1.Actuators.FeedValve_AV4x101.cmdClose.DOut', pin_4A5E1556A870DE8E := 'RES0.Reactor1.Actuators.LowerLevelValve_AV4x102.cmdOpen.DOut', pin_BB019F781B1BA10A := 'RES0.Reactor1.Actuators.LowerLevelValve_AV4x102.cmdClose.DOut', pin_86F66632C3A9C16C := 'RES0.Reactor1.Actuators.DischargeValve_AV4x103.cmdOpen.DOut', pin_B6D2486BB09D13CD := 'RES0.Reactor1.Actuators.DischargeValve_AV4x103.cmdClose.DOut', pin_51993B782C6727EF := 'RES0.Reactor2.Actuators.VentAerationGridValve_AV4x107.cmdOpen.DOut', pin_C59E5F7297A9D375 := 'RES0.Reactor2.Actuators.VentAerationGridValve_AV4x107.cmdClose.DOut', pin_713D841585687888 := 'RES0.Reactor2.Actuators.AirFillValveSludgeDischarge_AV4x171.cmdOpen.DOut', pin_F178B2FCFCB541E9 := 'RES0.Reactor2.Actuators.AirFillValveSludgeDischarge_AV4x171.cmdClose.DOut');
        A8_DQ32TK0 : IO_DQ32(pin_302C3F69182ABC91 := '$${PATH}A8_DQ32TK_WORD0', pin_449EC30B868089F7 := '$${PATH}A8_DQ32TK_WORD1', pin_4CB528AC475AE599 := 'RES0.A3_DI32K0.A3_DI32K0_CONN', pin_9A3A1A81B7B6D445 := 'RES0.Reactor2.Actuators.VentSludgeGridValve_AV4x172.cmdOpen.DOut', pin_574F19B312039273 := 'RES0.Reactor2.Actuators.VentSludgeGridValve_AV4x172.cmdClose.DOut', pin_289462D1695B79B9 := 'RES0.Reactor2.Actuators.FeedValve_AV4x101.cmdOpen.DOut', pin_312C400F6E937723 := 'RES0.Reactor2.Actuators.FeedValve_AV4x101.cmdClose.DOut', pin_3BE637AB2D7945FF := 'RES0.Reactor2.Actuators.LowerLevelValve_AV4x102.cmdOpen.DOut', pin_22A55DF5D197312F := 'RES0.Reactor2.Actuators.LowerLevelValve_AV4x102.cmdClose.DOut', pin_8561E9473423D106 := 'RES0.Reactor2.Actuators.DischargeValve_AV4x103.cmdOpen.DOut', pin_22A9D026EB73BE1F := 'RES0.Reactor2.Actuators.DischargeValve_AV4x103.cmdClose.DOut', pin_FA96DB2F4BA1237E := 'RES0.SludgeBuffer.Actuators.ValveSupernatantReturn.cmdOpen.DOut', pin_29C78CF381382FF2 := 'RES0.SludgeBuffer.Actuators.ValveSupernatantReturn.cmdClose.DOut', pin_29CEA3759F3752DE := 'RES0.SludgeBuffer.Actuators.ValveBuffer.cmdOpen.DOut', pin_886E7CBF7859CEF7 := 'RES0.SludgeBuffer.Actuators.ValveBuffer.cmdClose.DOut', pin_FD4664BC008BF5D6 := 'RES0.SludgeBuffer.Actuators.ValveInfeed.cmdOpen.DOut', pin_33252EF2B10EEA13 := 'RES0.SludgeBuffer.Actuators.ValveInfeed.cmdClose.DOut', pin_0AA04E78B7312E60 := 'RES0.SludgeBuffer.Actuators.ValveTank2.cmdOpen.DOut', pin_753BEBC4FB000D5B := 'RES0.SludgeBuffer.Actuators.ValveTank2.cmdClose.DOut', pin_9E16F3DA85027DF7 := 'RES0.SludgeBuffer.Actuators.ValveTank1.cmdOpen.DOut', pin_3452F813357567DB := 'RES0.SludgeBuffer.Actuators.ValveTank1.cmdClose.DOut', pin_19CF596687475EFF := 'RES0.Reactor1.Actuators.AerationBlockValve_AV4x170.cmdOpen.DOut', pin_894AD674E7043530 := 'RES0.Reactor1.Actuators.AerationBlockValve_AV4x170.cmdClose.DOut', pin_4C1794B9AC53DE50 := 'RES0.Reactor2.Actuators.AerationBlockValve_AV4x170.cmdOpen.DOut', pin_B27C16F31DA61BFA := 'RES0.Reactor2.Actuators.AerationBlockValve_AV4x170.cmdClose.DOut');
        SUB_A3_DI32K0 : IO_DI32(pin_46CCA44197086456 := '$${PATH}SUB_A3_DI32K_WORD0', pin_0CD1E891B208CBDA := '$${PATH}SUB_A3_DI32K_WORD1', pin_029A065AE8EEF4A5 := '$${PATH}SUB_A3_DI32K0_CONN', pin_23FCAB00EAAA7E55 := 'RES0.Aerator.Actuators.V4603.LocalPanel.PowerFb', pin_3F9A9A7D3F756840 := 'RES0.Aerator.Actuators.V4604.LocalPanel.PowerFb');
        SUB_A4_DI32K0 : IO_DI32(pin_46CCA44197086456 := '$${PATH}SUB_A4_DI32K_WORD0', pin_0CD1E891B208CBDA := '$${PATH}SUB_A4_DI32K_WORD1', pin_029A065AE8EEF4A5 := 'RES0.SUB_A3_DI32K0.SUB_A3_DI32K0_CONN', pin_3B4E2202D2B578AA := 'RES0.Aerator.Actuators.V4601.LocalPanel.PowerFb', pin_C8A2275FCD06007F := 'RES0.Aerator.Actuators.V4602.LocalPanel.PowerFb');
        SUB_A6_DI32K0 : IO_DI32(pin_46CCA44197086456 := '$${PATH}SUB_A6_DI32K_WORD0', pin_0CD1E891B208CBDA := '$${PATH}SUB_A6_DI32K_WORD1', pin_029A065AE8EEF4A5 := 'RES0.SUB_A3_DI32K0.SUB_A3_DI32K0_CONN', pin_255156C9E2C187C7 := 'RES0.Aerator.Actuators.AV46_001.fbOpen.DIn', pin_A4FEA1DCF2974931 := 'RES0.Aerator.Actuators.AV46_001.fbClose.DIn', pin_330A6B5BAE9F40D2 := 'RES0.Aerator.Actuators.AV46_002.fbOpen.DIn', pin_341ABC323332EA3F := 'RES0.Aerator.Actuators.AV46_002.fbClose.DIn', pin_15A3E3BB9AE8E740 := 'RES0.Aerator.Actuators.AV46_003.fbOpen.DIn', pin_6F381A44E74CF961 := 'RES0.Aerator.Actuators.AV46_003.fbClose.DIn', pin_28174C1DE6948A82 := 'RES0.Aerator.Actuators.AV46_012.fbOpen.DIn', pin_1BA632E0922A0983 := 'RES0.Aerator.Actuators.AV46_012.fbClose.DIn', pin_23FCAB00EAAA7E55 := 'RES0.Aerator.Actuators.AV46_022.fbOpen.DIn', pin_3F9A9A7D3F756840 := 'RES0.Aerator.Actuators.AV46_022.fbClose.DIn', pin_7C7DB6F90D480DE8 := 'RES0.Aerator.Actuators.AV46_032.fbOpen.DIn', pin_E8D93A7BE9BA26AB := 'RES0.Aerator.Actuators.AV46_032.fbClose.DIn', pin_2C3BA8CD03BB1AD1 := 'RES0.Aerator.Actuators.AV46_042.fbOpen.DIn', pin_BD4DD77DC1DECA3F := 'RES0.Aerator.Actuators.AV46_042.fbClose.DIn');
        SUB_A8_DQ32TK0 : IO_DQ32(pin_302C3F69182ABC91 := '$${PATH}SUB_A8_DQ32TK_WORD0', pin_449EC30B868089F7 := '$${PATH}SUB_A8_DQ32TK_WORD1', pin_4CB528AC475AE599 := 'RES0.SUB_A3_DI32K0.SUB_A3_DI32K0_CONN', pin_19CF596687475EFF := 'RES0.Aerator.Actuators.AV46_001.cmdOpen.DOut', pin_894AD674E7043530 := 'RES0.Aerator.Actuators.AV46_001.cmdClose.DOut', pin_4C1794B9AC53DE50 := 'RES0.Aerator.Actuators.AV46_002.cmdOpen.DOut', pin_B27C16F31DA61BFA := 'RES0.Aerator.Actuators.AV46_002.cmdClose.DOut', pin_6AEF80E82895335D := 'RES0.Aerator.Actuators.AV46_003.cmdOpen.DOut', pin_4CE944D399950301 := 'RES0.Aerator.Actuators.AV46_003.cmdClose.DOut', pin_4A5E1556A870DE8E := 'RES0.Aerator.Actuators.AV46_012.cmdOpen.DOut', pin_BB019F781B1BA10A := 'RES0.Aerator.Actuators.AV46_012.cmdClose.DOut', pin_86F66632C3A9C16C := 'RES0.Aerator.Actuators.AV46_022.cmdOpen.DOut', pin_B6D2486BB09D13CD := 'RES0.Aerator.Actuators.AV46_022.cmdClose.DOut', pin_51993B782C6727EF := 'RES0.Aerator.Actuators.AV46_032.cmdOpen.DOut', pin_C59E5F7297A9D375 := 'RES0.Aerator.Actuators.AV46_032.cmdClose.DOut', pin_713D841585687888 := 'RES0.Aerator.Actuators.AV46_042.cmdOpen.DOut', pin_F178B2FCFCB541E9 := 'RES0.Aerator.Actuators.AV46_042.cmdClose.DOut');
        V4601_STS0 : IO_DI32(pin_46CCA44197086456 := '$${PATH}V4601_STATUS', pin_0CD1E891B208CBDA := '$${PATH}V4601_FAULT', pin_029A065AE8EEF4A5 := '$${PATH}V4601_CONN', pin_21F6274CBA1014D4 := 'RES0.Aerator.Actuators.V4601.LocalPanel.RemoteSelect', pin_828C0F18BDE4203E := 'RES0.Aerator.Actuators.V4601.fbFwd.DIn', pin_36419F0327C5E289 := 'RES0.Aerator.Actuators.V4601.LocalPanel.FrequencyInverterFail', pin_4067F611C03C22ED := 'RES0.Aerator.Actuators.V4601.LocalPanel.AtvReady');
        V4601_CMD0 : IO_DQ32(pin_302C3F69182ABC91 := '$${PATH}V4601_CMD_WORD', pin_449EC30B868089F7 := '$${PATH}V4601_WORD1_NAO_USADA', pin_9A3A1A81B7B6D445 := 'RES0.Aerator.Actuators.V4601.cmdFwd.DOut', pin_289462D1695B79B9 := 'RES0.Aerator.Actuators.V4601.LocalPanel.ResetError_ATV');
        V4602_STS0 : IO_DI32(pin_46CCA44197086456 := '$${PATH}V4602_STATUS', pin_0CD1E891B208CBDA := '$${PATH}V4602_FAULT', pin_029A065AE8EEF4A5 := '$${PATH}V4602_CONN', pin_21F6274CBA1014D4 := 'RES0.Aerator.Actuators.V4602.LocalPanel.RemoteSelect', pin_828C0F18BDE4203E := 'RES0.Aerator.Actuators.V4602.fbFwd.DIn', pin_36419F0327C5E289 := 'RES0.Aerator.Actuators.V4602.LocalPanel.FrequencyInverterFail', pin_4067F611C03C22ED := 'RES0.Aerator.Actuators.V4602.LocalPanel.AtvReady');
        V4602_CMD0 : IO_DQ32(pin_302C3F69182ABC91 := '$${PATH}V4602_CMD_WORD', pin_449EC30B868089F7 := '$${PATH}V4602_WORD1_NAO_USADA', pin_9A3A1A81B7B6D445 := 'RES0.Aerator.Actuators.V4602.cmdFwd.DOut', pin_289462D1695B79B9 := 'RES0.Aerator.Actuators.V4602.LocalPanel.ResetError_ATV');
        V4603_STS0 : IO_DI32(pin_46CCA44197086456 := '$${PATH}V4603_STATUS', pin_0CD1E891B208CBDA := '$${PATH}V4603_FAULT', pin_029A065AE8EEF4A5 := '$${PATH}V4603_CONN', pin_21F6274CBA1014D4 := 'RES0.Aerator.Actuators.V4603.LocalPanel.RemoteSelect', pin_828C0F18BDE4203E := 'RES0.Aerator.Actuators.V4603.fbFwd.DIn', pin_36419F0327C5E289 := 'RES0.Aerator.Actuators.V4603.LocalPanel.FrequencyInverterFail', pin_4067F611C03C22ED := 'RES0.Aerator.Actuators.V4603.LocalPanel.AtvReady');
        V4603_CMD0 : IO_DQ32(pin_302C3F69182ABC91 := '$${PATH}V4603_CMD_WORD', pin_449EC30B868089F7 := '$${PATH}V4603_WORD1_NAO_USADA', pin_9A3A1A81B7B6D445 := 'RES0.Aerator.Actuators.V4603.cmdFwd.DOut', pin_289462D1695B79B9 := 'RES0.Aerator.Actuators.V4603.LocalPanel.ResetError_ATV');
        V4604_STS0 : IO_DI32(pin_46CCA44197086456 := '$${PATH}V4604_STATUS', pin_0CD1E891B208CBDA := '$${PATH}V4604_FAULT', pin_029A065AE8EEF4A5 := '$${PATH}V4604_CONN', pin_21F6274CBA1014D4 := 'RES0.Aerator.Actuators.V4604.LocalPanel.RemoteSelect', pin_828C0F18BDE4203E := 'RES0.Aerator.Actuators.V4604.fbFwd.DIn', pin_36419F0327C5E289 := 'RES0.Aerator.Actuators.V4604.LocalPanel.FrequencyInverterFail', pin_4067F611C03C22ED := 'RES0.Aerator.Actuators.V4604.LocalPanel.AtvReady');
        V4604_CMD0 : IO_DQ32(pin_302C3F69182ABC91 := '$${PATH}V4604_CMD_WORD', pin_449EC30B868089F7 := '$${PATH}V4604_WORD1_NAO_USADA', pin_9A3A1A81B7B6D445 := 'RES0.Aerator.Actuators.V4604.cmdFwd.DOut', pin_289462D1695B79B9 := 'RES0.Aerator.Actuators.V4604.LocalPanel.ResetError_ATV');
        SludgeHoldingTank1 : SludgeHoldingTank;
        SludgeHoldingTank2 : SludgeHoldingTank;
      END_FBS
      EVENT_CONNECTIONS
        START.COLD TO DPAC_FULLINIT1.INIT;
        START.WARM TO DPAC_FULLINIT1.INIT;
        START.ONLINECHANGE TO DPAC_FULLINIT1.OC_RETRIGGER;
      END_CONNECTIONS
      ADAPTER_CONNECTIONS
        EmergencyManagement.5C1263F1F6F0F578 TO EmergencyReactor1.73503C83163B2D86;
        EmergencyManagement.6B6FC4EBFE551754 TO EmergencyReactor2.73503C83163B2D86;
        OTHERS_DISCHARGE_VALVES_FB.00DDB30B96836B1C TO Reactor2.AE9DB11716461BE5;
        Reactor2.53509993DCC2E69E TO EmergencyManagement.8D40980BCD10D06B;
        Reactor2.E962C7AC1C669349 TO Aerator.036B0699AE92B07E;
        EmergencyReactor2.ADE9AC252194767E TO Reactor2.4FE3E9A63522A043;
        SludgeBuffer.F8A56E33E99EA0E4 TO Reactor2.64A5E847CFF537B2;
        EmergencyReactor2.D6CF55AACA664FB9 TO EmergencySB.A9597B321AC24B8F;
        EmergencyReactor1.D6CF55AACA664FB9 TO EmergencySB.E201588BE0264C59;
        OTHERS_DISCHARGE_VALVES_FB.82A979F8A1C1CE4A TO Reactor1.AE9DB11716461BE5;
        Reactor1.53509993DCC2E69E TO EmergencyManagement.03E1DF24854B5087;
        Reactor1.E962C7AC1C669349 TO Aerator.IBlowerReactor;
        EmergencyReactor1.ADE9AC252194767E TO Reactor1.4FE3E9A63522A043;
        SludgeBuffer.5220CD4AB4D5EF57 TO Reactor1.64A5E847CFF537B2;
        Mode.39 TO Reactor1.8E8BC8CAE0ABBEF0;
        Mode.40 TO Reactor2.8E8BC8CAE0ABBEF0;
        Mode.55 TO EmergencyManagement.FA37C5C7FF880AB4;
        InfluentFeed.06B5BF90025137D8 TO SludgeBuffer.04BD059D1BCDA8FF;
        InfluentFeed.08DA021DBE2FF670 TO SludgeBuffer.34E82C716D68805B;
        Reactor1.EF12C2F0857E0401 TO InfluentFeed.458126F8619187E9;
        Reactor2.EF12C2F0857E0401 TO InfluentFeed.13A00CB3B1B3C5BD;
        SludgeBuffer.2EF6B69B645AE6E1 TO InfluentFeed.9135BA3E72B25810;
        InfluentFeed.072EC58E32F5B902 TO Reactor1.9D6CC0A1E886795A;
        InfluentFeed.57887779F0B6E332 TO Reactor2.9D6CC0A1E886795A;
        SludgeHoldingTank1.745E7C7F86CD93D6 TO SludgeBuffer.1369AAF8C65D025F;
        SludgeHoldingTank2.745E7C7F86CD93D6 TO SludgeBuffer.103390B72A3B733A;
        EmergencyManagement.10001B393681040B TO OTHERS_DISCHARGE_VALVES_FB.0FC638121CDA6752;
        SludgeBuffer.8B97DDD2DF3E853F TO EmergencyManagement.92B17EFA7CB0DA14;
        HeartBeat1.40 TO Mode.6E012D59F948069E;
        Mode.50 TO SludgeBuffer.6D7943A09F73313C;
        SludgeBuffer.0CE6DD66A1C58D5B TO Reactor1.6D054A47338EC161;
        SludgeBuffer.DE069E6752438E1A TO Reactor2.6D054A47338EC161;
        EmergencySB.CC52284A3E90E837 TO SludgeBuffer.8642DEF89CD05FB2;
      END_CONNECTIONS
    END_RESOURCE
  END_DEVICE
  DEVICE HMI : HMI_NET
  END_DEVICE
  DEVICE HMI_NEREDA : HMI_NET
  END_DEVICE
  MAPPINGS
    Hidryco_Application.OpenWebPage ON M262_Nereda.RES0;
    Hidryco_Application.OTHERS_DISCHARGE_VALVES_FB ON M262_Nereda.RES0;
    Hidryco_Application.EmergencyManagement ON M262_Nereda.RES0;
    Hidryco_Application.Utilities ON M262_Nereda.RES0;
    Hidryco_Application.EnergySignal ON M262_Nereda.RES0;
    Hidryco_Application.HeartBeat1 ON M262_Nereda.RES0;
    Hidryco_Application.Aerator ON M262_Nereda.RES0;
    Hidryco_Application.SludgeBuffer ON M262_Nereda.RES0;
    Hidryco_Application.EmergencyReactor1 ON M262_Nereda.RES0;
    Hidryco_Application.EmergencyReactor2 ON M262_Nereda.RES0;
    Hidryco_Application.Reactor2 ON M262_Nereda.RES0;
    Hidryco_Application.EmergencySB ON M262_Nereda.RES0;
    Hidryco_Application.Reactor1 ON M262_Nereda.RES0;
    Hidryco_Application.Mode ON M262_Nereda.RES0;
    Hidryco_Application.InfluentFeed ON M262_Nereda.RES0;
    Hidryco_Application.A3_DI32K0 ON M262_Nereda.RES0;
    Hidryco_Application.A4_DI32K0 ON M262_Nereda.RES0;
    Hidryco_Application.A5_DI32K0 ON M262_Nereda.RES0;
    Hidryco_Application.A6_DI32K0 ON M262_Nereda.RES0;
    Hidryco_Application.A7_DQ32TK0 ON M262_Nereda.RES0;
    Hidryco_Application.A8_DQ32TK0 ON M262_Nereda.RES0;
    Hidryco_Application.SUB_A3_DI32K0 ON M262_Nereda.RES0;
    Hidryco_Application.SUB_A4_DI32K0 ON M262_Nereda.RES0;
    Hidryco_Application.SUB_A6_DI32K0 ON M262_Nereda.RES0;
    Hidryco_Application.SUB_A8_DQ32TK0 ON M262_Nereda.RES0;
    Hidryco_Application.V4601_STS0 ON M262_Nereda.RES0;
    Hidryco_Application.V4601_CMD0 ON M262_Nereda.RES0;
    Hidryco_Application.V4602_STS0 ON M262_Nereda.RES0;
    Hidryco_Application.V4602_CMD0 ON M262_Nereda.RES0;
    Hidryco_Application.V4603_STS0 ON M262_Nereda.RES0;
    Hidryco_Application.V4603_CMD0 ON M262_Nereda.RES0;
    Hidryco_Application.V4604_STS0 ON M262_Nereda.RES0;
    Hidryco_Application.V4604_CMD0 ON M262_Nereda.RES0;
    Hidryco_Application.SludgeHoldingTank1 ON M262_Nereda.RES0;
    Hidryco_Application.SludgeHoldingTank2 ON M262_Nereda.RES0;
  END_MAPPINGS
END_SYSTEM
(* other elements stored in the file *)
(* Layer Name=ETE_TJ *)
(* FrameName Name=FRAME9 *)
(* FrameName Name=FRAME11 *)
(* Layer Name=IOs *)
(* FBName Name=A3_DI32K0 *)
(* FBName Name=A4_DI32K0 *)
(* FBName Name=A5_DI32K0 *)
(* FBName Name=A6_DI32K0 *)
(* FBName Name=A7_DQ32TK0 *)
(* FBName Name=A8_DQ32TK0 *)
(* FBName Name=SUB_A3_DI32K0 *)
(* FBName Name=SUB_A4_DI32K0 *)
(* FBName Name=SUB_A6_DI32K0 *)
(* FBName Name=SUB_A8_DQ32TK0 *)
(* FBName Name=V4601_STS0 *)
(* FBName Name=V4601_CMD0 *)
(* FBName Name=V4602_STS0 *)
(* FBName Name=V4602_CMD0 *)
(* FBName Name=V4603_STS0 *)
(* FBName Name=V4603_CMD0 *)
(* FBName Name=V4604_STS0 *)
(* FBName Name=V4604_CMD0 *)
(* DefaultLayer Name=Nereda *)
